Staubli VAL3: stop.pgx

program stop()
begin
  cls()
  title("")
end
